PROGRAM prgRWLynus
VAR
	fbRW1		: FB_ReadWrite;
	fbRW2		: FB_ReadWrite;
	fbRW3		: FB_ReadWrite;
	fbRW4		: FB_ReadWrite;
	fbRW5		: FB_ReadWrite;
	fbRW6		: FB_ReadWrite;
END_VAR

fbRW1();
fbRW2();
fbRW3();
fbRW4();
fbRW5();
fbRW6();

END_PROGRAM

(* stored: Version 1.1.0.1, ProductVersion 3.1.4024.9
   POU prgRWLynus: Id {62995b61-8431-4bff-affc-05b4805b57ee}, SpecialFunc None *)
